// Mitsubishi GX Developer project: PLC_PCO520L2   PLC: Q06UDEH

PROGRAM ALARM
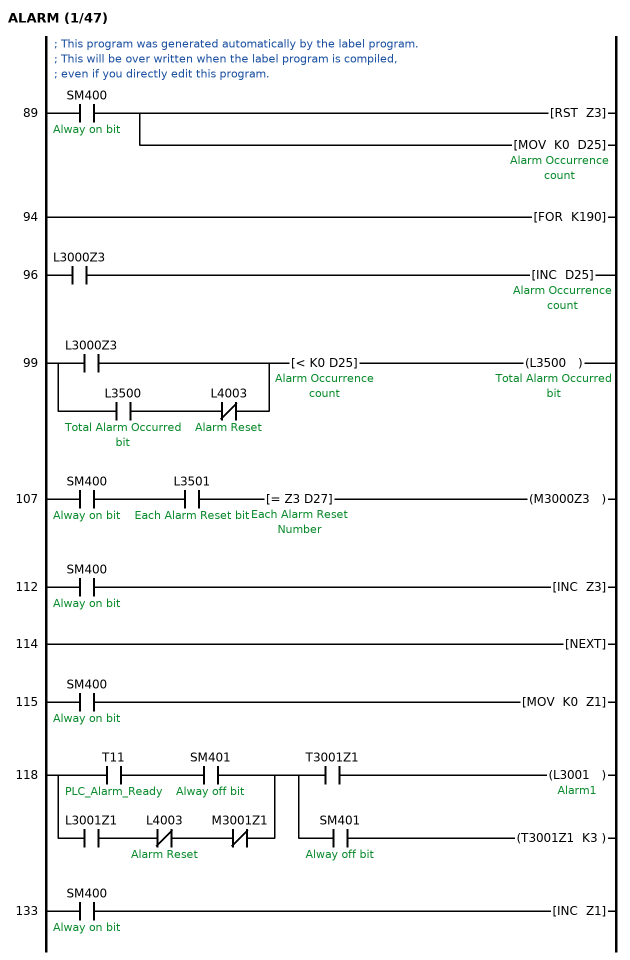
; This program was generated automatically by the label program.
; This will be over written when the label program is compiled,
; even if you directly edit this program.
89    LD      SM400  ; Alway on bit
      RST     Z3
      MOV     K0 D25  ; Alarm Occurrence count
94    FOR     K190
96    LD      L3000Z3
      INC     D25
99    LD      L3000Z3
      LD      L3500  ; Total Alarm Occurred bit
      ANI     L4003  ; Alarm Reset
      ORB
      AND<    K0 D25  ; Alarm Occurrence count
      OUT     L3500  ; Total Alarm Occurred bit
107   LD      SM400  ; Alway on bit
      AND     L3501  ; Each Alarm Reset bit
      AND=    Z3 D27  ; Each Alarm Reset Number
      OUT     M3000Z3
112   LD      SM400  ; Alway on bit
      INC     Z3
114   NEXT
115   LD      SM400  ; Alway on bit
      MOV     K0 Z1
118   LD      T11  ; PLC_Alarm_Ready
      AND     SM401  ; Alway off bit
      LD      L3001Z1
      ANI     L4003  ; Alarm Reset
      ANI     M3001Z1
      ORB
      MPS
      AND     T3001Z1
      OUT     L3001  ; Alarm1
      MPP
      AND     SM401  ; Alway off bit
      OUT     T3001Z1 K3
133   LD      SM400  ; Alway on bit
      INC     Z1
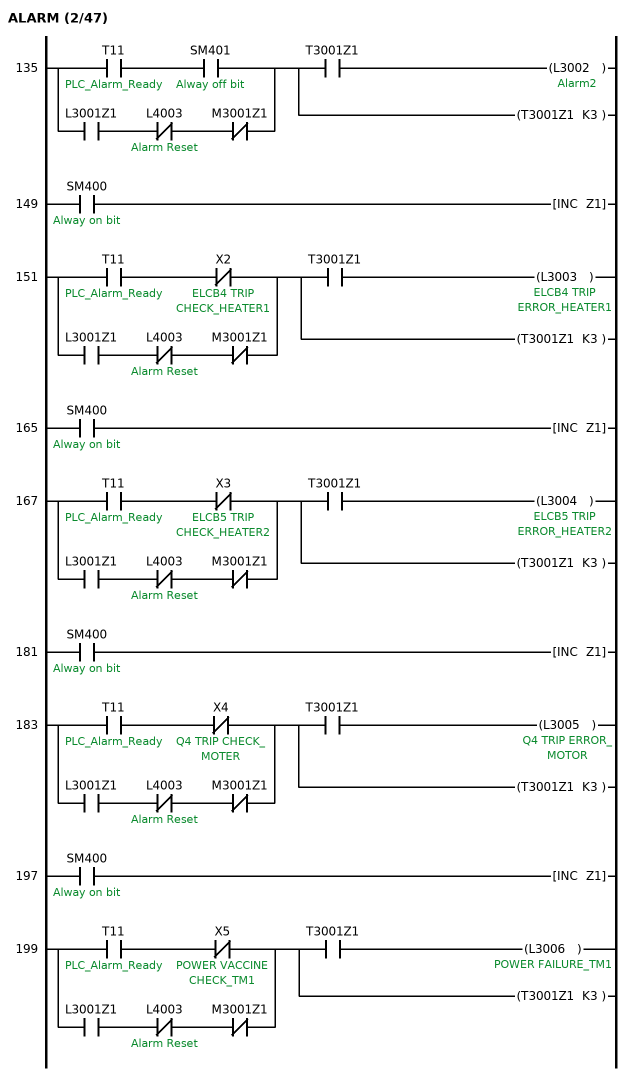
135   LD      T11  ; PLC_Alarm_Ready
      AND     SM401  ; Alway off bit
      LD      L3001Z1
      ANI     L4003  ; Alarm Reset
      ANI     M3001Z1
      ORB
      MPS
      AND     T3001Z1
      OUT     L3002  ; Alarm2
      MPP
      OUT     T3001Z1 K3
149   LD      SM400  ; Alway on bit
      INC     Z1
151   LD      T11  ; PLC_Alarm_Ready
      ANI     X2  ; ELCB4 TRIP CHECK_HEATER1
      LD      L3001Z1
      ANI     L4003  ; Alarm Reset
      ANI     M3001Z1
      ORB
      MPS
      AND     T3001Z1
      OUT     L3003  ; ELCB4 TRIP ERROR_HEATER1
      MPP
      OUT     T3001Z1 K3
165   LD      SM400  ; Alway on bit
      INC     Z1
167   LD      T11  ; PLC_Alarm_Ready
      ANI     X3  ; ELCB5 TRIP CHECK_HEATER2
      LD      L3001Z1
      ANI     L4003  ; Alarm Reset
      ANI     M3001Z1
      ORB
      MPS
      AND     T3001Z1
      OUT     L3004  ; ELCB5 TRIP ERROR_HEATER2
      MPP
      OUT     T3001Z1 K3
181   LD      SM400  ; Alway on bit
      INC     Z1
183   LD      T11  ; PLC_Alarm_Ready
      ANI     X4  ; Q4 TRIP CHECK_MOTER
      LD      L3001Z1
      ANI     L4003  ; Alarm Reset
      ANI     M3001Z1
      ORB
      MPS
      AND     T3001Z1
      OUT     L3005  ; Q4 TRIP ERROR_MOTOR
      MPP
      OUT     T3001Z1 K3
197   LD      SM400  ; Alway on bit
      INC     Z1
199   LD      T11  ; PLC_Alarm_Ready
      ANI     X5  ; POWER VACCINE CHECK_TM1
      LD      L3001Z1
      ANI     L4003  ; Alarm Reset
      ANI     M3001Z1
      ORB
      MPS
      AND     T3001Z1
      OUT     L3006  ; POWER FAILURE_TM1
      MPP
      OUT     T3001Z1 K3
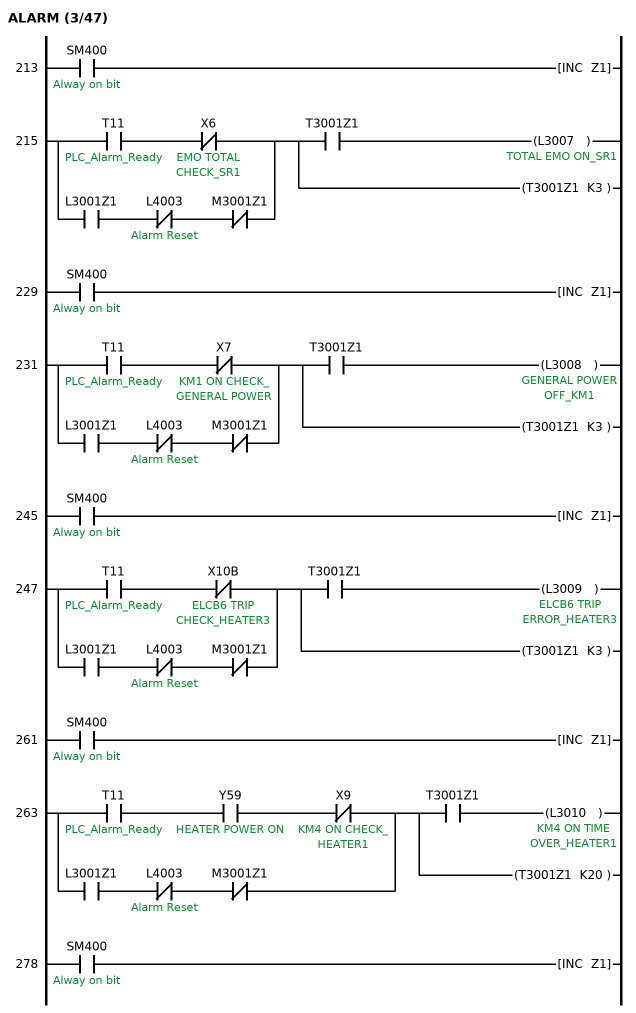
213   LD      SM400  ; Alway on bit
      INC     Z1
215   LD      T11  ; PLC_Alarm_Ready
      ANI     X6  ; EMO TOTAL CHECK_SR1
      LD      L3001Z1
      ANI     L4003  ; Alarm Reset
      ANI     M3001Z1
      ORB
      MPS
      AND     T3001Z1
      OUT     L3007  ; TOTAL EMO ON_SR1
      MPP
      OUT     T3001Z1 K3
229   LD      SM400  ; Alway on bit
      INC     Z1
231   LD      T11  ; PLC_Alarm_Ready
      ANI     X7  ; KM1 ON CHECK_GENERAL POWER
      LD      L3001Z1
      ANI     L4003  ; Alarm Reset
      ANI     M3001Z1
      ORB
      MPS
      AND     T3001Z1
      OUT     L3008  ; GENERAL POWER OFF_KM1
      MPP
      OUT     T3001Z1 K3
245   LD      SM400  ; Alway on bit
      INC     Z1
247   LD      T11  ; PLC_Alarm_Ready
      ANI     X10B  ; ELCB6 TRIP CHECK_HEATER3
      LD      L3001Z1
      ANI     L4003  ; Alarm Reset
      ANI     M3001Z1
      ORB
      MPS
      AND     T3001Z1
      OUT     L3009  ; ELCB6 TRIP ERROR_HEATER3
      MPP
      OUT     T3001Z1 K3
261   LD      SM400  ; Alway on bit
      INC     Z1
263   LD      T11  ; PLC_Alarm_Ready
      AND     Y59  ; HEATER POWER ON
      ANI     X9  ; KM4 ON CHECK_HEATER1
      LD      L3001Z1
      ANI     L4003  ; Alarm Reset
      ANI     M3001Z1
      ORB
      MPS
      AND     T3001Z1
      OUT     L3010  ; KM4 ON TIME OVER_HEATER1
      MPP
      OUT     T3001Z1 K20
278   LD      SM400  ; Alway on bit
      INC     Z1
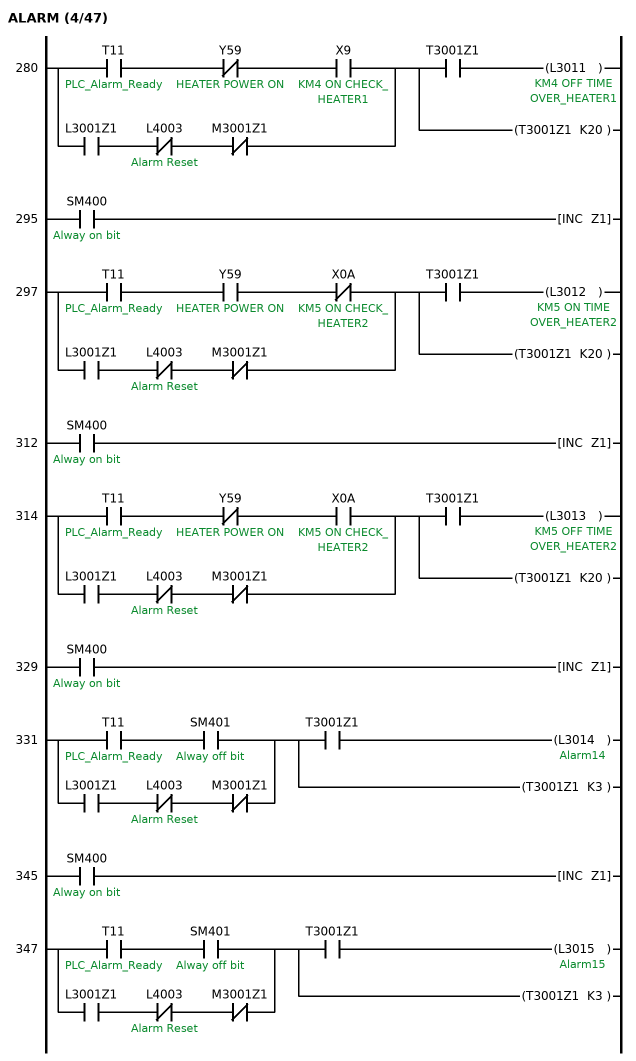
280   LD      T11  ; PLC_Alarm_Ready
      ANI     Y59  ; HEATER POWER ON
      AND     X9  ; KM4 ON CHECK_HEATER1
      LD      L3001Z1
      ANI     L4003  ; Alarm Reset
      ANI     M3001Z1
      ORB
      MPS
      AND     T3001Z1
      OUT     L3011  ; KM4 OFF TIME OVER_HEATER1
      MPP
      OUT     T3001Z1 K20
295   LD      SM400  ; Alway on bit
      INC     Z1
297   LD      T11  ; PLC_Alarm_Ready
      AND     Y59  ; HEATER POWER ON
      ANI     X0A  ; KM5 ON CHECK_HEATER2
      LD      L3001Z1
      ANI     L4003  ; Alarm Reset
      ANI     M3001Z1
      ORB
      MPS
      AND     T3001Z1
      OUT     L3012  ; KM5 ON TIME OVER_HEATER2
      MPP
      OUT     T3001Z1 K20
312   LD      SM400  ; Alway on bit
      INC     Z1
314   LD      T11  ; PLC_Alarm_Ready
      ANI     Y59  ; HEATER POWER ON
      AND     X0A  ; KM5 ON CHECK_HEATER2
      LD      L3001Z1
      ANI     L4003  ; Alarm Reset
      ANI     M3001Z1
      ORB
      MPS
      AND     T3001Z1
      OUT     L3013  ; KM5 OFF TIME OVER_HEATER2
      MPP
      OUT     T3001Z1 K20
329   LD      SM400  ; Alway on bit
      INC     Z1
331   LD      T11  ; PLC_Alarm_Ready
      AND     SM401  ; Alway off bit
      LD      L3001Z1
      ANI     L4003  ; Alarm Reset
      ANI     M3001Z1
      ORB
      MPS
      AND     T3001Z1
      OUT     L3014  ; Alarm14
      MPP
      OUT     T3001Z1 K3
345   LD      SM400  ; Alway on bit
      INC     Z1
347   LD      T11  ; PLC_Alarm_Ready
      AND     SM401  ; Alway off bit
      LD      L3001Z1
      ANI     L4003  ; Alarm Reset
      ANI     M3001Z1
      ORB
      MPS
      AND     T3001Z1
      OUT     L3015  ; Alarm15
      MPP
      OUT     T3001Z1 K3
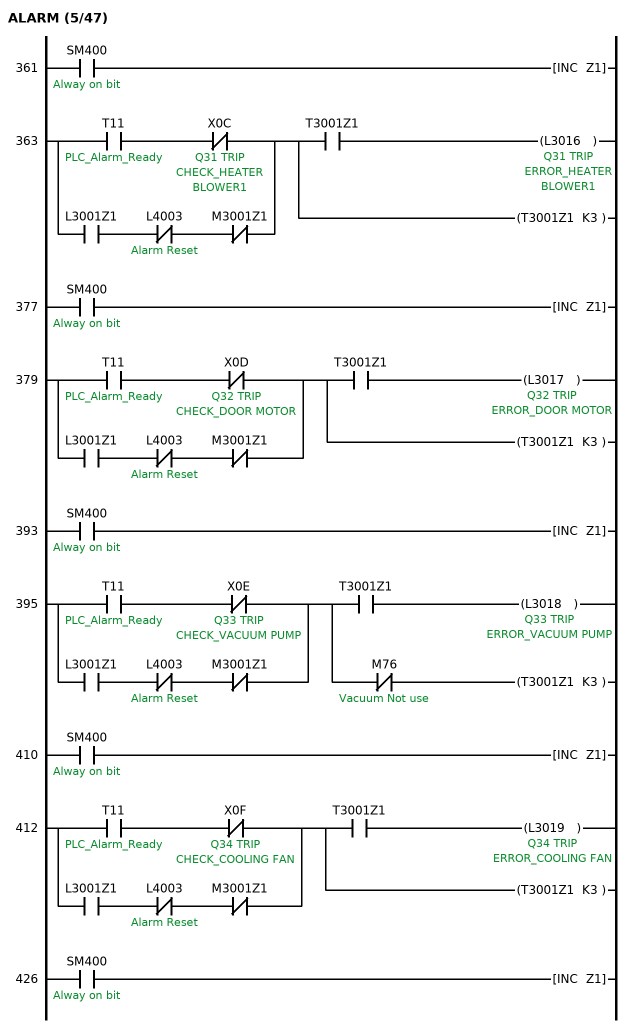
361   LD      SM400  ; Alway on bit
      INC     Z1
363   LD      T11  ; PLC_Alarm_Ready
      ANI     X0C  ; Q31 TRIP CHECK_HEATER BLOWER1
      LD      L3001Z1
      ANI     L4003  ; Alarm Reset
      ANI     M3001Z1
      ORB
      MPS
      AND     T3001Z1
      OUT     L3016  ; Q31 TRIP ERROR_HEATER BLOWER1
      MPP
      OUT     T3001Z1 K3
377   LD      SM400  ; Alway on bit
      INC     Z1
379   LD      T11  ; PLC_Alarm_Ready
      ANI     X0D  ; Q32 TRIP CHECK_DOOR MOTOR
      LD      L3001Z1
      ANI     L4003  ; Alarm Reset
      ANI     M3001Z1
      ORB
      MPS
      AND     T3001Z1
      OUT     L3017  ; Q32 TRIP ERROR_DOOR MOTOR
      MPP
      OUT     T3001Z1 K3
393   LD      SM400  ; Alway on bit
      INC     Z1
395   LD      T11  ; PLC_Alarm_Ready
      ANI     X0E  ; Q33 TRIP CHECK_VACUUM PUMP
      LD      L3001Z1
      ANI     L4003  ; Alarm Reset
      ANI     M3001Z1
      ORB
      MPS
      AND     T3001Z1
      OUT     L3018  ; Q33 TRIP ERROR_VACUUM PUMP
      MPP
      ANI     M76  ; Vacuum Not use
      OUT     T3001Z1 K3
410   LD      SM400  ; Alway on bit
      INC     Z1
412   LD      T11  ; PLC_Alarm_Ready
      ANI     X0F  ; Q34 TRIP CHECK_COOLING FAN
      LD      L3001Z1
      ANI     L4003  ; Alarm Reset
      ANI     M3001Z1
      ORB
      MPS
      AND     T3001Z1
      OUT     L3019  ; Q34 TRIP ERROR_COOLING FAN
      MPP
      OUT     T3001Z1 K3
426   LD      SM400  ; Alway on bit
      INC     Z1
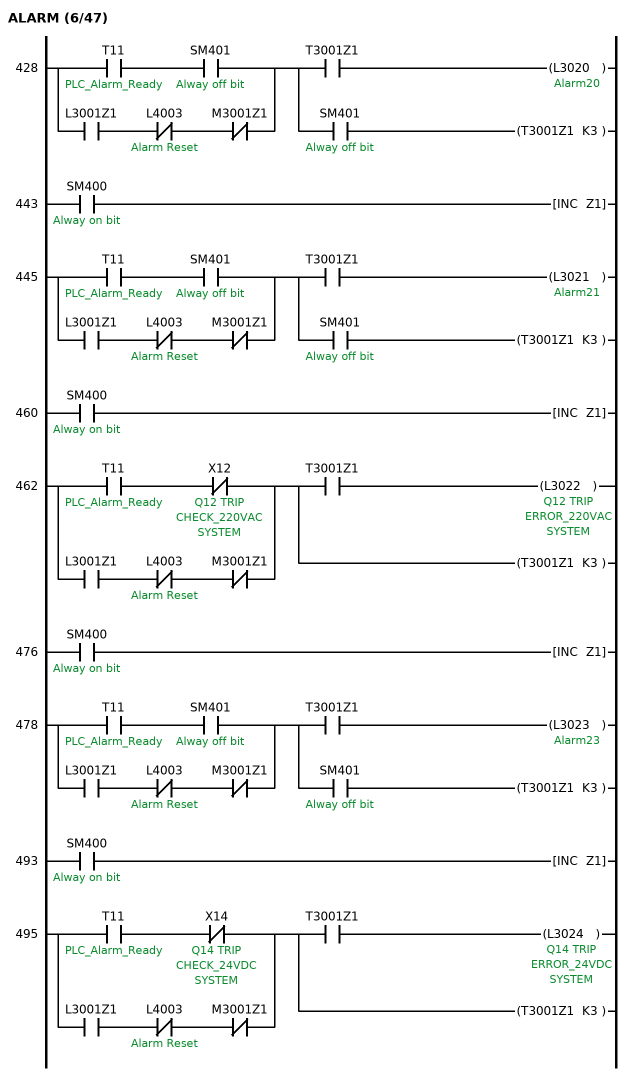
428   LD      T11  ; PLC_Alarm_Ready
      AND     SM401  ; Alway off bit
      LD      L3001Z1
      ANI     L4003  ; Alarm Reset
      ANI     M3001Z1
      ORB
      MPS
      AND     T3001Z1
      OUT     L3020  ; Alarm20
      MPP
      AND     SM401  ; Alway off bit
      OUT     T3001Z1 K3
443   LD      SM400  ; Alway on bit
      INC     Z1
445   LD      T11  ; PLC_Alarm_Ready
      AND     SM401  ; Alway off bit
      LD      L3001Z1
      ANI     L4003  ; Alarm Reset
      ANI     M3001Z1
      ORB
      MPS
      AND     T3001Z1
      OUT     L3021  ; Alarm21
      MPP
      AND     SM401  ; Alway off bit
      OUT     T3001Z1 K3
460   LD      SM400  ; Alway on bit
      INC     Z1
462   LD      T11  ; PLC_Alarm_Ready
      ANI     X12  ; Q12 TRIP CHECK_220VAC SYSTEM
      LD      L3001Z1
      ANI     L4003  ; Alarm Reset
      ANI     M3001Z1
      ORB
      MPS
      AND     T3001Z1
      OUT     L3022  ; Q12 TRIP ERROR_220VAC SYSTEM
      MPP
      OUT     T3001Z1 K3
476   LD      SM400  ; Alway on bit
      INC     Z1
478   LD      T11  ; PLC_Alarm_Ready
      AND     SM401  ; Alway off bit
      LD      L3001Z1
      ANI     L4003  ; Alarm Reset
      ANI     M3001Z1
      ORB
      MPS
      AND     T3001Z1
      OUT     L3023  ; Alarm23
      MPP
      AND     SM401  ; Alway off bit
      OUT     T3001Z1 K3
493   LD      SM400  ; Alway on bit
      INC     Z1
495   LD      T11  ; PLC_Alarm_Ready
      ANI     X14  ; Q14 TRIP CHECK_24VDC SYSTEM
      LD      L3001Z1
      ANI     L4003  ; Alarm Reset
      ANI     M3001Z1
      ORB
      MPS
      AND     T3001Z1
      OUT     L3024  ; Q14 TRIP ERROR_24VDC SYSTEM
      MPP
      OUT     T3001Z1 K3
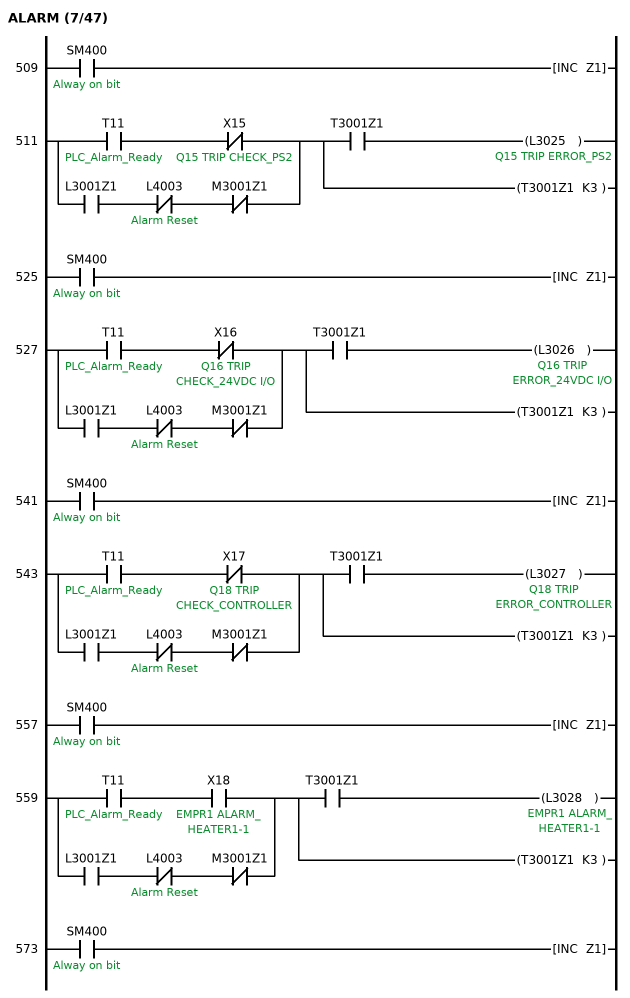
509   LD      SM400  ; Alway on bit
      INC     Z1
511   LD      T11  ; PLC_Alarm_Ready
      ANI     X15  ; Q15 TRIP CHECK_PS2
      LD      L3001Z1
      ANI     L4003  ; Alarm Reset
      ANI     M3001Z1
      ORB
      MPS
      AND     T3001Z1
      OUT     L3025  ; Q15 TRIP ERROR_PS2
      MPP
      OUT     T3001Z1 K3
525   LD      SM400  ; Alway on bit
      INC     Z1
527   LD      T11  ; PLC_Alarm_Ready
      ANI     X16  ; Q16 TRIP CHECK_24VDC I/O
      LD      L3001Z1
      ANI     L4003  ; Alarm Reset
      ANI     M3001Z1
      ORB
      MPS
      AND     T3001Z1
      OUT     L3026  ; Q16 TRIP ERROR_24VDC I/O
      MPP
      OUT     T3001Z1 K3
541   LD      SM400  ; Alway on bit
      INC     Z1
543   LD      T11  ; PLC_Alarm_Ready
      ANI     X17  ; Q18 TRIP CHECK_CONTROLLER
      LD      L3001Z1
      ANI     L4003  ; Alarm Reset
      ANI     M3001Z1
      ORB
      MPS
      AND     T3001Z1
      OUT     L3027  ; Q18 TRIP ERROR_CONTROLLER
      MPP
      OUT     T3001Z1 K3
557   LD      SM400  ; Alway on bit
      INC     Z1
559   LD      T11  ; PLC_Alarm_Ready
      AND     X18  ; EMPR1 ALARM_HEATER1-1
      LD      L3001Z1
      ANI     L4003  ; Alarm Reset
      ANI     M3001Z1
      ORB
      MPS
      AND     T3001Z1
      OUT     L3028  ; EMPR1 ALARM_HEATER1-1
      MPP
      OUT     T3001Z1 K3
573   LD      SM400  ; Alway on bit
      INC     Z1
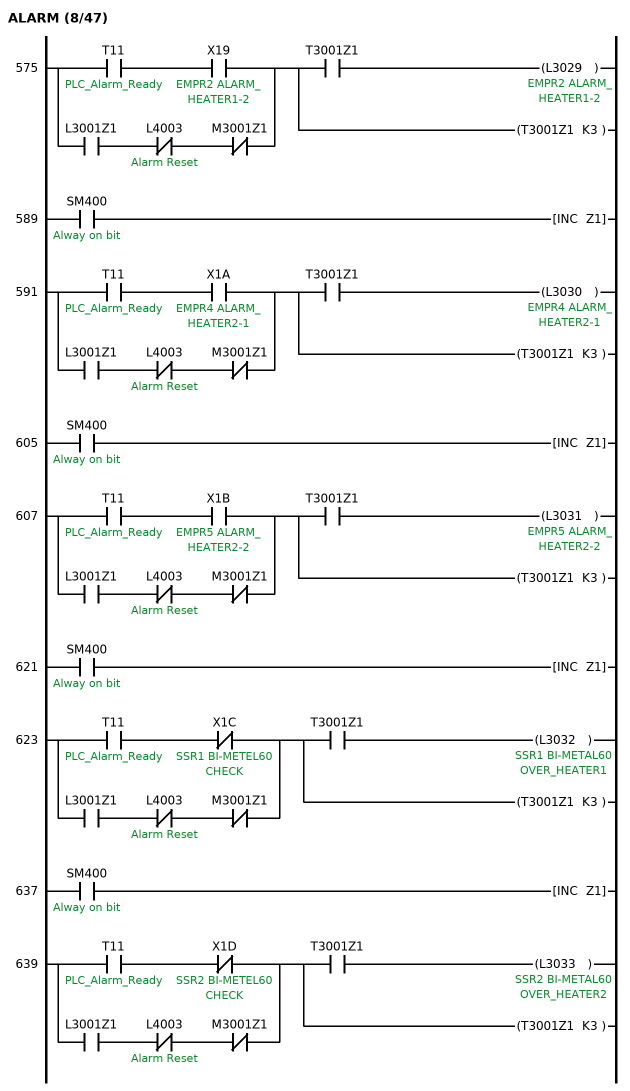
575   LD      T11  ; PLC_Alarm_Ready
      AND     X19  ; EMPR2 ALARM_HEATER1-2
      LD      L3001Z1
      ANI     L4003  ; Alarm Reset
      ANI     M3001Z1
      ORB
      MPS
      AND     T3001Z1
      OUT     L3029  ; EMPR2 ALARM_HEATER1-2
      MPP
      OUT     T3001Z1 K3
589   LD      SM400  ; Alway on bit
      INC     Z1
591   LD      T11  ; PLC_Alarm_Ready
      AND     X1A  ; EMPR4 ALARM_HEATER2-1
      LD      L3001Z1
      ANI     L4003  ; Alarm Reset
      ANI     M3001Z1
      ORB
      MPS
      AND     T3001Z1
      OUT     L3030  ; EMPR4 ALARM_HEATER2-1
      MPP
      OUT     T3001Z1 K3
605   LD      SM400  ; Alway on bit
      INC     Z1
607   LD      T11  ; PLC_Alarm_Ready
      AND     X1B  ; EMPR5 ALARM_HEATER2-2
      LD      L3001Z1
      ANI     L4003  ; Alarm Reset
      ANI     M3001Z1
      ORB
      MPS
      AND     T3001Z1
      OUT     L3031  ; EMPR5 ALARM_HEATER2-2
      MPP
      OUT     T3001Z1 K3
621   LD      SM400  ; Alway on bit
      INC     Z1
623   LD      T11  ; PLC_Alarm_Ready
      ANI     X1C  ; SSR1 BI-METEL60 CHECK
      LD      L3001Z1
      ANI     L4003  ; Alarm Reset
      ANI     M3001Z1
      ORB
      MPS
      AND     T3001Z1
      OUT     L3032  ; SSR1 BI-METAL60 OVER_HEATER1
      MPP
      OUT     T3001Z1 K3
637   LD      SM400  ; Alway on bit
      INC     Z1
639   LD      T11  ; PLC_Alarm_Ready
      ANI     X1D  ; SSR2 BI-METEL60 CHECK
      LD      L3001Z1
      ANI     L4003  ; Alarm Reset
      ANI     M3001Z1
      ORB
      MPS
      AND     T3001Z1
      OUT     L3033  ; SSR2 BI-METAL60 OVER_HEATER2
      MPP
      OUT     T3001Z1 K3
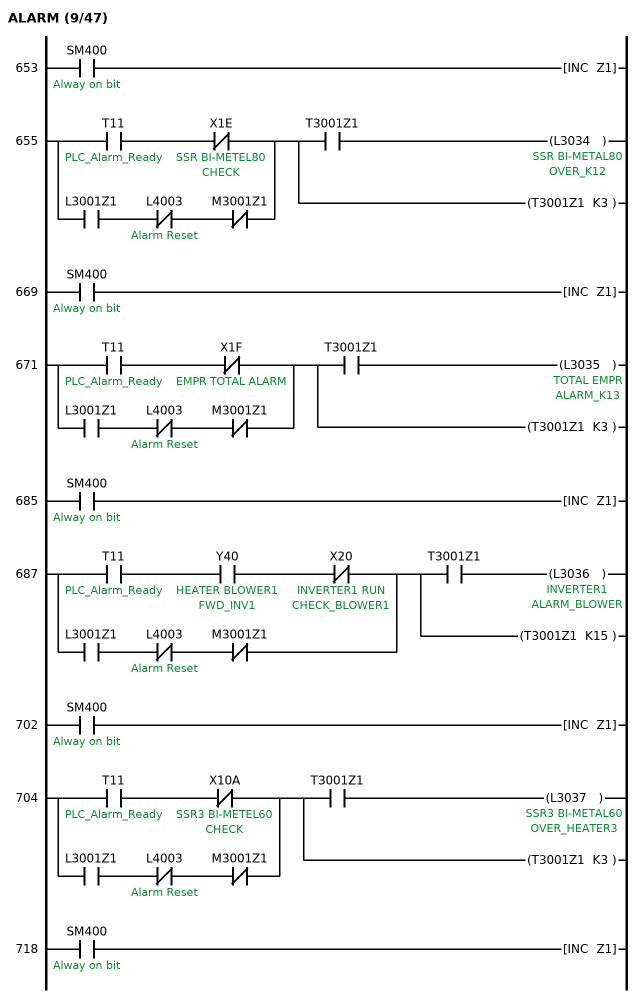
653   LD      SM400  ; Alway on bit
      INC     Z1
655   LD      T11  ; PLC_Alarm_Ready
      ANI     X1E  ; SSR BI-METEL80 CHECK
      LD      L3001Z1
      ANI     L4003  ; Alarm Reset
      ANI     M3001Z1
      ORB
      MPS
      AND     T3001Z1
      OUT     L3034  ; SSR BI-METAL80 OVER_K12
      MPP
      OUT     T3001Z1 K3
669   LD      SM400  ; Alway on bit
      INC     Z1
671   LD      T11  ; PLC_Alarm_Ready
      ANI     X1F  ; EMPR TOTAL ALARM
      LD      L3001Z1
      ANI     L4003  ; Alarm Reset
      ANI     M3001Z1
      ORB
      MPS
      AND     T3001Z1
      OUT     L3035  ; TOTAL EMPR ALARM_K13
      MPP
      OUT     T3001Z1 K3
685   LD      SM400  ; Alway on bit
      INC     Z1
687   LD      T11  ; PLC_Alarm_Ready
      AND     Y40  ; HEATER BLOWER1 FWD_INV1
      ANI     X20  ; INVERTER1 RUN CHECK_BLOWER1
      LD      L3001Z1
      ANI     L4003  ; Alarm Reset
      ANI     M3001Z1
      ORB
      MPS
      AND     T3001Z1
      OUT     L3036  ; INVERTER1 ALARM_BLOWER
      MPP
      OUT     T3001Z1 K15
702   LD      SM400  ; Alway on bit
      INC     Z1
704   LD      T11  ; PLC_Alarm_Ready
      ANI     X10A  ; SSR3 BI-METEL60 CHECK
      LD      L3001Z1
      ANI     L4003  ; Alarm Reset
      ANI     M3001Z1
      ORB
      MPS
      AND     T3001Z1
      OUT     L3037  ; SSR3 BI-METAL60 OVER_HEATER3
      MPP
      OUT     T3001Z1 K3
718   LD      SM400  ; Alway on bit
      INC     Z1
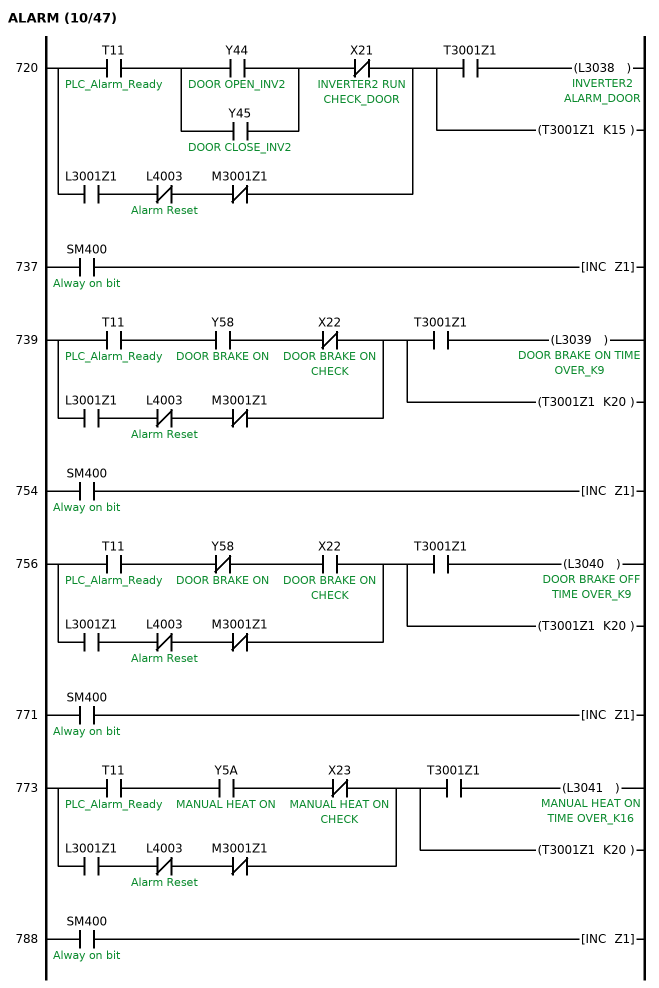
720   LD      T11  ; PLC_Alarm_Ready
      LD      Y44  ; DOOR OPEN_INV2
      OR      Y45  ; DOOR CLOSE_INV2
      ANB
      ANI     X21  ; INVERTER2 RUN CHECK_DOOR
      LD      L3001Z1
      ANI     L4003  ; Alarm Reset
      ANI     M3001Z1
      ORB
      MPS
      AND     T3001Z1
      OUT     L3038  ; INVERTER2 ALARM_DOOR
      MPP
      OUT     T3001Z1 K15
737   LD      SM400  ; Alway on bit
      INC     Z1
739   LD      T11  ; PLC_Alarm_Ready
      AND     Y58  ; DOOR BRAKE ON
      ANI     X22  ; DOOR BRAKE ON CHECK
      LD      L3001Z1
      ANI     L4003  ; Alarm Reset
      ANI     M3001Z1
      ORB
      MPS
      AND     T3001Z1
      OUT     L3039  ; DOOR BRAKE ON TIME OVER_K9
      MPP
      OUT     T3001Z1 K20
754   LD      SM400  ; Alway on bit
      INC     Z1
756   LD      T11  ; PLC_Alarm_Ready
      ANI     Y58  ; DOOR BRAKE ON
      AND     X22  ; DOOR BRAKE ON CHECK
      LD      L3001Z1
      ANI     L4003  ; Alarm Reset
      ANI     M3001Z1
      ORB
      MPS
      AND     T3001Z1
      OUT     L3040  ; DOOR BRAKE OFF TIME OVER_K9
      MPP
      OUT     T3001Z1 K20
771   LD      SM400  ; Alway on bit
      INC     Z1
773   LD      T11  ; PLC_Alarm_Ready
      AND     Y5A  ; MANUAL HEAT ON
      ANI     X23  ; MANUAL HEAT ON CHECK
      LD      L3001Z1
      ANI     L4003  ; Alarm Reset
      ANI     M3001Z1
      ORB
      MPS
      AND     T3001Z1
      OUT     L3041  ; MANUAL HEAT ON TIME OVER_K16
      MPP
      OUT     T3001Z1 K20
788   LD      SM400  ; Alway on bit
      INC     Z1
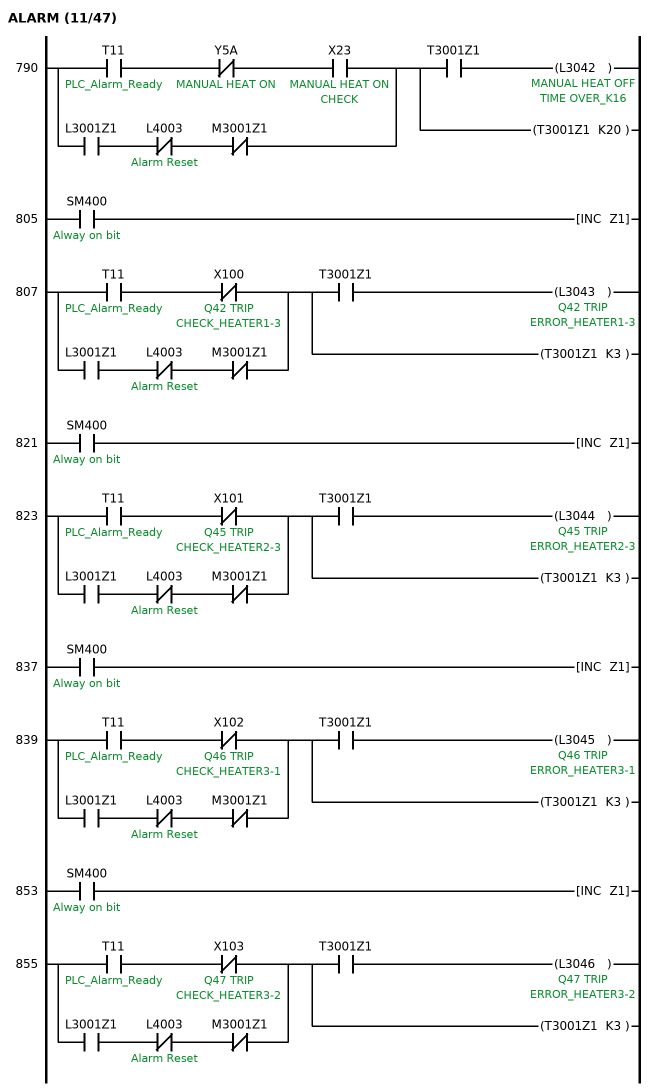
790   LD      T11  ; PLC_Alarm_Ready
      ANI     Y5A  ; MANUAL HEAT ON
      AND     X23  ; MANUAL HEAT ON CHECK
      LD      L3001Z1
      ANI     L4003  ; Alarm Reset
      ANI     M3001Z1
      ORB
      MPS
      AND     T3001Z1
      OUT     L3042  ; MANUAL HEAT OFF TIME OVER_K16
      MPP
      OUT     T3001Z1 K20
805   LD      SM400  ; Alway on bit
      INC     Z1
807   LD      T11  ; PLC_Alarm_Ready
      ANI     X100  ; Q42 TRIP CHECK_HEATER1-3
      LD      L3001Z1
      ANI     L4003  ; Alarm Reset
      ANI     M3001Z1
      ORB
      MPS
      AND     T3001Z1
      OUT     L3043  ; Q42 TRIP ERROR_HEATER1-3
      MPP
      OUT     T3001Z1 K3
821   LD      SM400  ; Alway on bit
      INC     Z1
823   LD      T11  ; PLC_Alarm_Ready
      ANI     X101  ; Q45 TRIP CHECK_HEATER2-3
      LD      L3001Z1
      ANI     L4003  ; Alarm Reset
      ANI     M3001Z1
      ORB
      MPS
      AND     T3001Z1
      OUT     L3044  ; Q45 TRIP ERROR_HEATER2-3
      MPP
      OUT     T3001Z1 K3
837   LD      SM400  ; Alway on bit
      INC     Z1
839   LD      T11  ; PLC_Alarm_Ready
      ANI     X102  ; Q46 TRIP CHECK_HEATER3-1
      LD      L3001Z1
      ANI     L4003  ; Alarm Reset
      ANI     M3001Z1
      ORB
      MPS
      AND     T3001Z1
      OUT     L3045  ; Q46 TRIP ERROR_HEATER3-1
      MPP
      OUT     T3001Z1 K3
853   LD      SM400  ; Alway on bit
      INC     Z1
855   LD      T11  ; PLC_Alarm_Ready
      ANI     X103  ; Q47 TRIP CHECK_HEATER3-2
      LD      L3001Z1
      ANI     L4003  ; Alarm Reset
      ANI     M3001Z1
      ORB
      MPS
      AND     T3001Z1
      OUT     L3046  ; Q47 TRIP ERROR_HEATER3-2
      MPP
      OUT     T3001Z1 K3
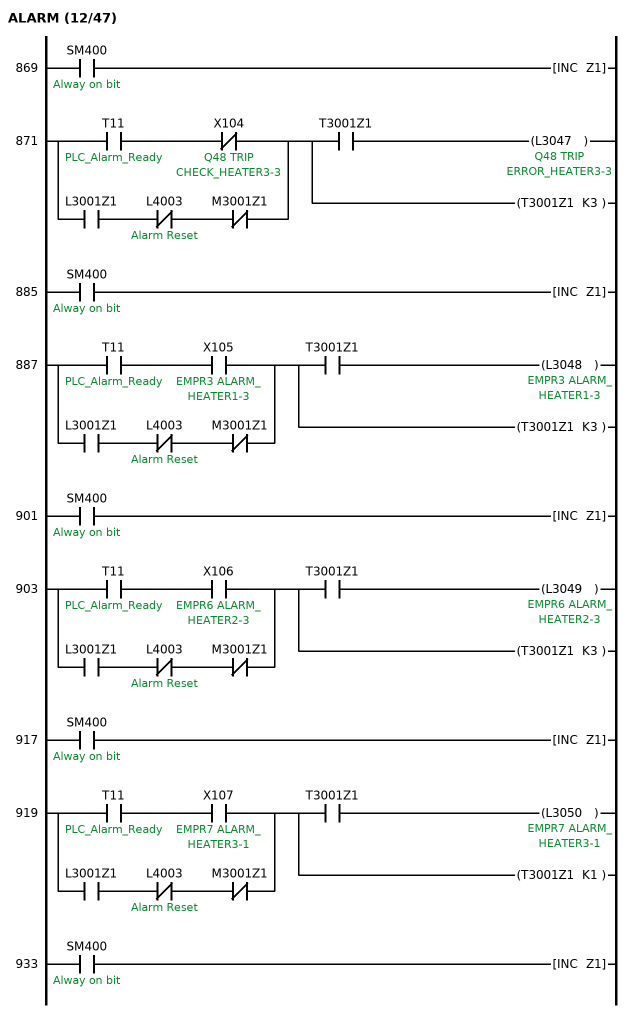
869   LD      SM400  ; Alway on bit
      INC     Z1
871   LD      T11  ; PLC_Alarm_Ready
      ANI     X104  ; Q48 TRIP CHECK_HEATER3-3
      LD      L3001Z1
      ANI     L4003  ; Alarm Reset
      ANI     M3001Z1
      ORB
      MPS
      AND     T3001Z1
      OUT     L3047  ; Q48 TRIP ERROR_HEATER3-3
      MPP
      OUT     T3001Z1 K3
885   LD      SM400  ; Alway on bit
      INC     Z1
887   LD      T11  ; PLC_Alarm_Ready
      AND     X105  ; EMPR3 ALARM_HEATER1-3
      LD      L3001Z1
      ANI     L4003  ; Alarm Reset
      ANI     M3001Z1
      ORB
      MPS
      AND     T3001Z1
      OUT     L3048  ; EMPR3 ALARM_HEATER1-3
      MPP
      OUT     T3001Z1 K3
901   LD      SM400  ; Alway on bit
      INC     Z1
903   LD      T11  ; PLC_Alarm_Ready
      AND     X106  ; EMPR6 ALARM_HEATER2-3
      LD      L3001Z1
      ANI     L4003  ; Alarm Reset
      ANI     M3001Z1
      ORB
      MPS
      AND     T3001Z1
      OUT     L3049  ; EMPR6 ALARM_HEATER2-3
      MPP
      OUT     T3001Z1 K3
917   LD      SM400  ; Alway on bit
      INC     Z1
919   LD      T11  ; PLC_Alarm_Ready
      AND     X107  ; EMPR7 ALARM_HEATER3-1
      LD      L3001Z1
      ANI     L4003  ; Alarm Reset
      ANI     M3001Z1
      ORB
      MPS
      AND     T3001Z1
      OUT     L3050  ; EMPR7 ALARM_HEATER3-1
      MPP
      OUT     T3001Z1 K1
933   LD      SM400  ; Alway on bit
      INC     Z1
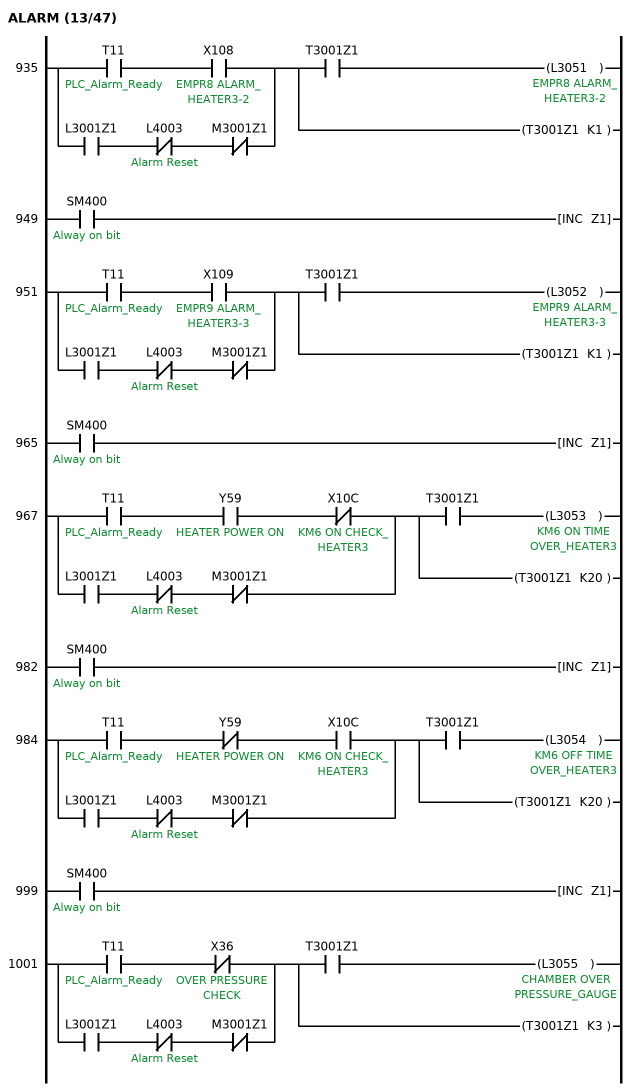
935   LD      T11  ; PLC_Alarm_Ready
      AND     X108  ; EMPR8 ALARM_HEATER3-2
      LD      L3001Z1
      ANI     L4003  ; Alarm Reset
      ANI     M3001Z1
      ORB
      MPS
      AND     T3001Z1
      OUT     L3051  ; EMPR8 ALARM_HEATER3-2
      MPP
      OUT     T3001Z1 K1
949   LD      SM400  ; Alway on bit
      INC     Z1
951   LD      T11  ; PLC_Alarm_Ready
      AND     X109  ; EMPR9 ALARM_HEATER3-3
      LD      L3001Z1
      ANI     L4003  ; Alarm Reset
      ANI     M3001Z1
      ORB
      MPS
      AND     T3001Z1
      OUT     L3052  ; EMPR9 ALARM_HEATER3-3
      MPP
      OUT     T3001Z1 K1
965   LD      SM400  ; Alway on bit
      INC     Z1
967   LD      T11  ; PLC_Alarm_Ready
      AND     Y59  ; HEATER POWER ON
      ANI     X10C  ; KM6 ON CHECK_HEATER3
      LD      L3001Z1
      ANI     L4003  ; Alarm Reset
      ANI     M3001Z1
      ORB
      MPS
      AND     T3001Z1
      OUT     L3053  ; KM6 ON TIME OVER_HEATER3
      MPP
      OUT     T3001Z1 K20
982   LD      SM400  ; Alway on bit
      INC     Z1
984   LD      T11  ; PLC_Alarm_Ready
      ANI     Y59  ; HEATER POWER ON
      AND     X10C  ; KM6 ON CHECK_HEATER3
      LD      L3001Z1
      ANI     L4003  ; Alarm Reset
      ANI     M3001Z1
      ORB
      MPS
      AND     T3001Z1
      OUT     L3054  ; KM6 OFF TIME OVER_HEATER3
      MPP
      OUT     T3001Z1 K20
999   LD      SM400  ; Alway on bit
      INC     Z1
1001  LD      T11  ; PLC_Alarm_Ready
      ANI     X36  ; OVER PRESSURE CHECK
      LD      L3001Z1
      ANI     L4003  ; Alarm Reset
      ANI     M3001Z1
      ORB
      MPS
      AND     T3001Z1
      OUT     L3055  ; CHAMBER OVER PRESSURE_GAUGE
      MPP
      OUT     T3001Z1 K3
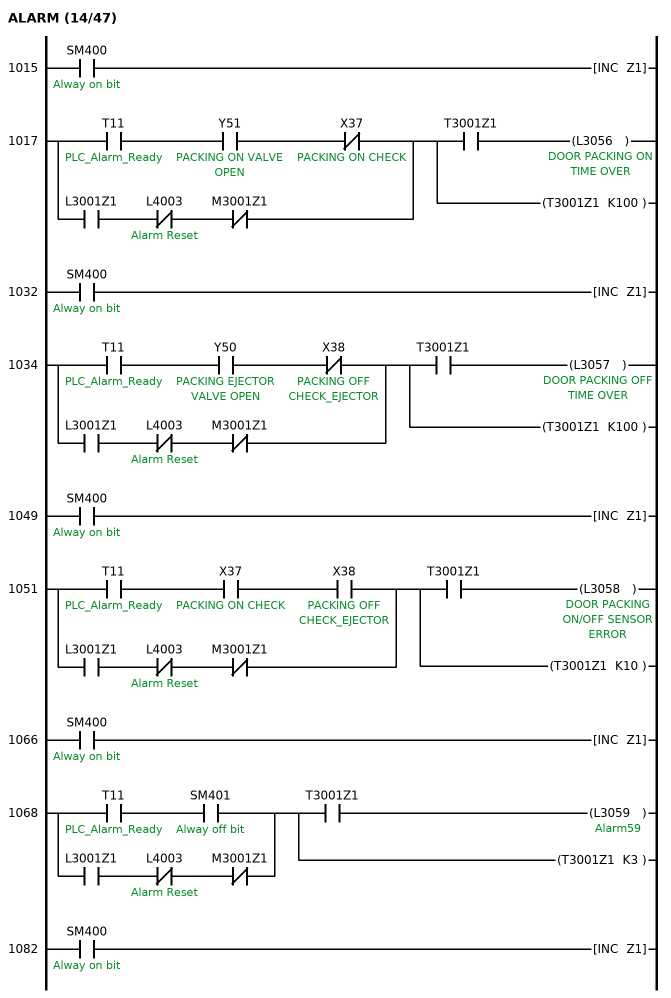
1015  LD      SM400  ; Alway on bit
      INC     Z1
1017  LD      T11  ; PLC_Alarm_Ready
      AND     Y51  ; PACKING ON VALVE OPEN
      ANI     X37  ; PACKING ON CHECK
      LD      L3001Z1
      ANI     L4003  ; Alarm Reset
      ANI     M3001Z1
      ORB
      MPS
      AND     T3001Z1
      OUT     L3056  ; DOOR PACKING ON TIME OVER
      MPP
      OUT     T3001Z1 K100
1032  LD      SM400  ; Alway on bit
      INC     Z1
1034  LD      T11  ; PLC_Alarm_Ready
      AND     Y50  ; PACKING EJECTOR VALVE OPEN
      ANI     X38  ; PACKING OFF CHECK_EJECTOR
      LD      L3001Z1
      ANI     L4003  ; Alarm Reset
      ANI     M3001Z1
      ORB
      MPS
      AND     T3001Z1
      OUT     L3057  ; DOOR PACKING OFF TIME OVER
      MPP
      OUT     T3001Z1 K100
1049  LD      SM400  ; Alway on bit
      INC     Z1
1051  LD      T11  ; PLC_Alarm_Ready
      AND     X37  ; PACKING ON CHECK
      AND     X38  ; PACKING OFF CHECK_EJECTOR
      LD      L3001Z1
      ANI     L4003  ; Alarm Reset
      ANI     M3001Z1
      ORB
      MPS
      AND     T3001Z1
      OUT     L3058  ; DOOR PACKING ON/OFF SENSOR ERROR
      MPP
      OUT     T3001Z1 K10
1066  LD      SM400  ; Alway on bit
      INC     Z1
1068  LD      T11  ; PLC_Alarm_Ready
      AND     SM401  ; Alway off bit
      LD      L3001Z1
      ANI     L4003  ; Alarm Reset
      ANI     M3001Z1
      ORB
      MPS
      AND     T3001Z1
      OUT     L3059  ; Alarm59
      MPP
      OUT     T3001Z1 K3
1082  LD      SM400  ; Alway on bit
      INC     Z1
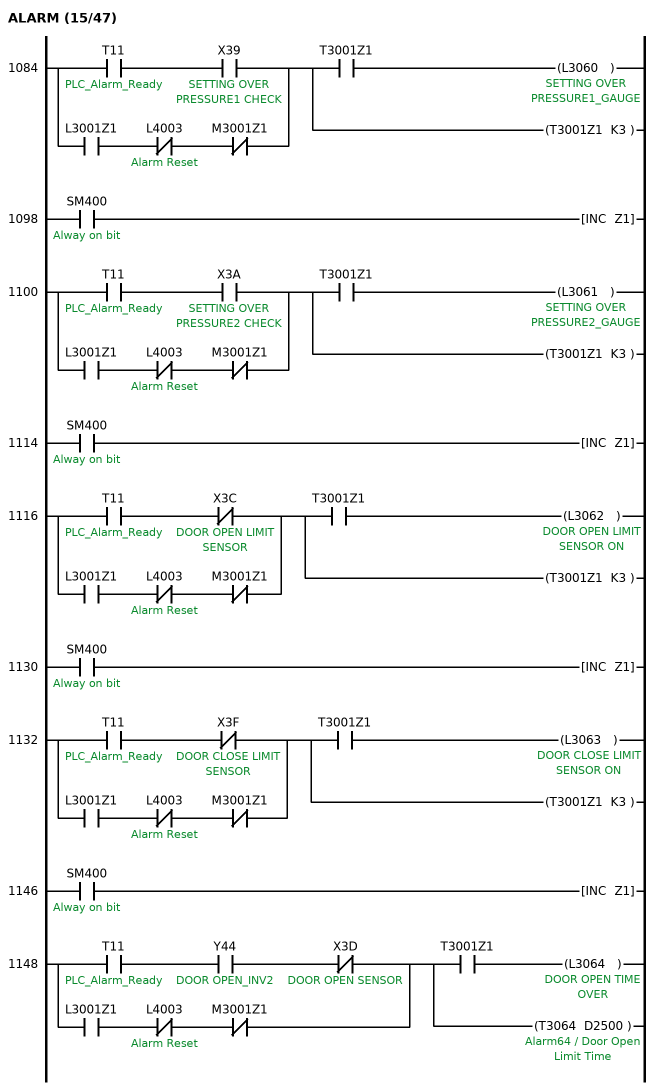
1084  LD      T11  ; PLC_Alarm_Ready
      AND     X39  ; SETTING OVER PRESSURE1 CHECK
      LD      L3001Z1
      ANI     L4003  ; Alarm Reset
      ANI     M3001Z1
      ORB
      MPS
      AND     T3001Z1
      OUT     L3060  ; SETTING OVER PRESSURE1_GAUGE
      MPP
      OUT     T3001Z1 K3
1098  LD      SM400  ; Alway on bit
      INC     Z1
1100  LD      T11  ; PLC_Alarm_Ready
      AND     X3A  ; SETTING OVER PRESSURE2 CHECK
      LD      L3001Z1
      ANI     L4003  ; Alarm Reset
      ANI     M3001Z1
      ORB
      MPS
      AND     T3001Z1
      OUT     L3061  ; SETTING OVER PRESSURE2_GAUGE
      MPP
      OUT     T3001Z1 K3
1114  LD      SM400  ; Alway on bit
      INC     Z1
1116  LD      T11  ; PLC_Alarm_Ready
      ANI     X3C  ; DOOR OPEN LIMIT SENSOR
      LD      L3001Z1
      ANI     L4003  ; Alarm Reset
      ANI     M3001Z1
      ORB
      MPS
      AND     T3001Z1
      OUT     L3062  ; DOOR OPEN LIMIT SENSOR ON
      MPP
      OUT     T3001Z1 K3
1130  LD      SM400  ; Alway on bit
      INC     Z1
1132  LD      T11  ; PLC_Alarm_Ready
      ANI     X3F  ; DOOR CLOSE LIMIT SENSOR
      LD      L3001Z1
      ANI     L4003  ; Alarm Reset
      ANI     M3001Z1
      ORB
      MPS
      AND     T3001Z1
      OUT     L3063  ; DOOR CLOSE LIMIT SENSOR ON
      MPP
      OUT     T3001Z1 K3
1146  LD      SM400  ; Alway on bit
      INC     Z1
1148  LD      T11  ; PLC_Alarm_Ready
      AND     Y44  ; DOOR OPEN_INV2
      ANI     X3D  ; DOOR OPEN SENSOR
      LD      L3001Z1
      ANI     L4003  ; Alarm Reset
      ANI     M3001Z1
      ORB
      MPS
      AND     T3001Z1
      OUT     L3064  ; DOOR OPEN TIME OVER
      MPP
      OUT     T3064 D2500  ; Alarm64 / Door Open Limit Time
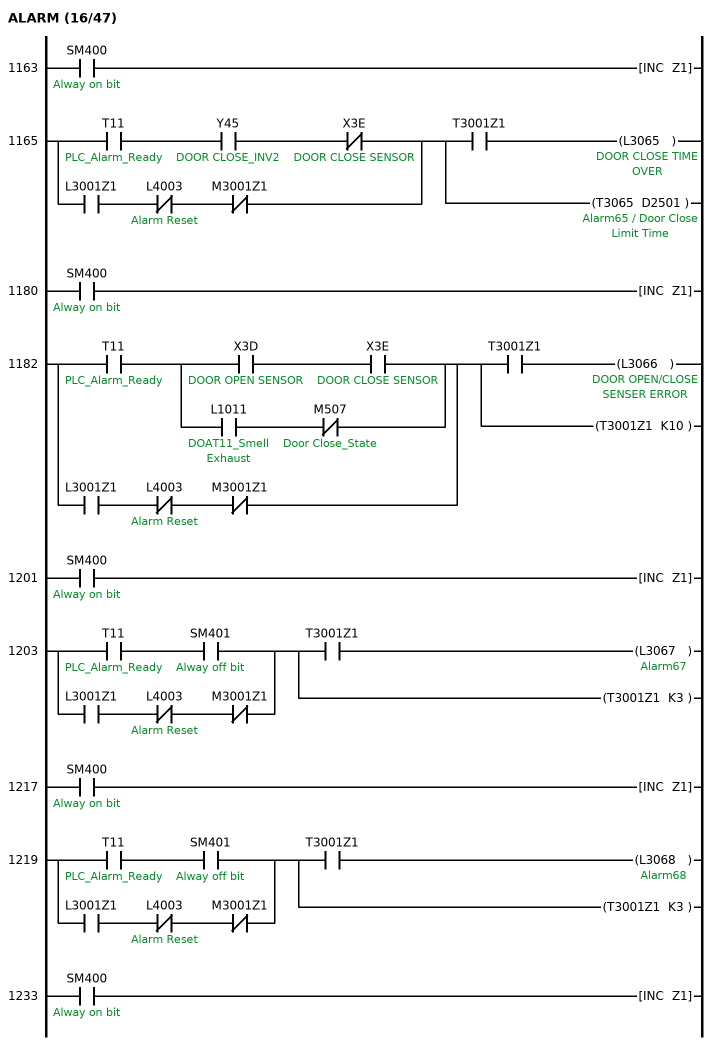
1163  LD      SM400  ; Alway on bit
      INC     Z1
1165  LD      T11  ; PLC_Alarm_Ready
      AND     Y45  ; DOOR CLOSE_INV2
      ANI     X3E  ; DOOR CLOSE SENSOR
      LD      L3001Z1
      ANI     L4003  ; Alarm Reset
      ANI     M3001Z1
      ORB
      MPS
      AND     T3001Z1
      OUT     L3065  ; DOOR CLOSE TIME OVER
      MPP
      OUT     T3065 D2501  ; Alarm65 / Door Close Limit Time
1180  LD      SM400  ; Alway on bit
      INC     Z1
1182  LD      T11  ; PLC_Alarm_Ready
      LD      X3D  ; DOOR OPEN SENSOR
      AND     X3E  ; DOOR CLOSE SENSOR
      LD      L1011  ; DOAT11_Smell Exhaust
      ANI     M507  ; Door Close_State
      ORB
      ANB
      LD      L3001Z1
      ANI     L4003  ; Alarm Reset
      ANI     M3001Z1
      ORB
      MPS
      AND     T3001Z1
      OUT     L3066  ; DOOR OPEN/CLOSE SENSER ERROR
      MPP
      OUT     T3001Z1 K10
1201  LD      SM400  ; Alway on bit
      INC     Z1
1203  LD      T11  ; PLC_Alarm_Ready
      AND     SM401  ; Alway off bit
      LD      L3001Z1
      ANI     L4003  ; Alarm Reset
      ANI     M3001Z1
      ORB
      MPS
      AND     T3001Z1
      OUT     L3067  ; Alarm67
      MPP
      OUT     T3001Z1 K3
1217  LD      SM400  ; Alway on bit
      INC     Z1
1219  LD      T11  ; PLC_Alarm_Ready
      AND     SM401  ; Alway off bit
      LD      L3001Z1
      ANI     L4003  ; Alarm Reset
      ANI     M3001Z1
      ORB
      MPS
      AND     T3001Z1
      OUT     L3068  ; Alarm68
      MPP
      OUT     T3001Z1 K3
1233  LD      SM400  ; Alway on bit
      INC     Z1
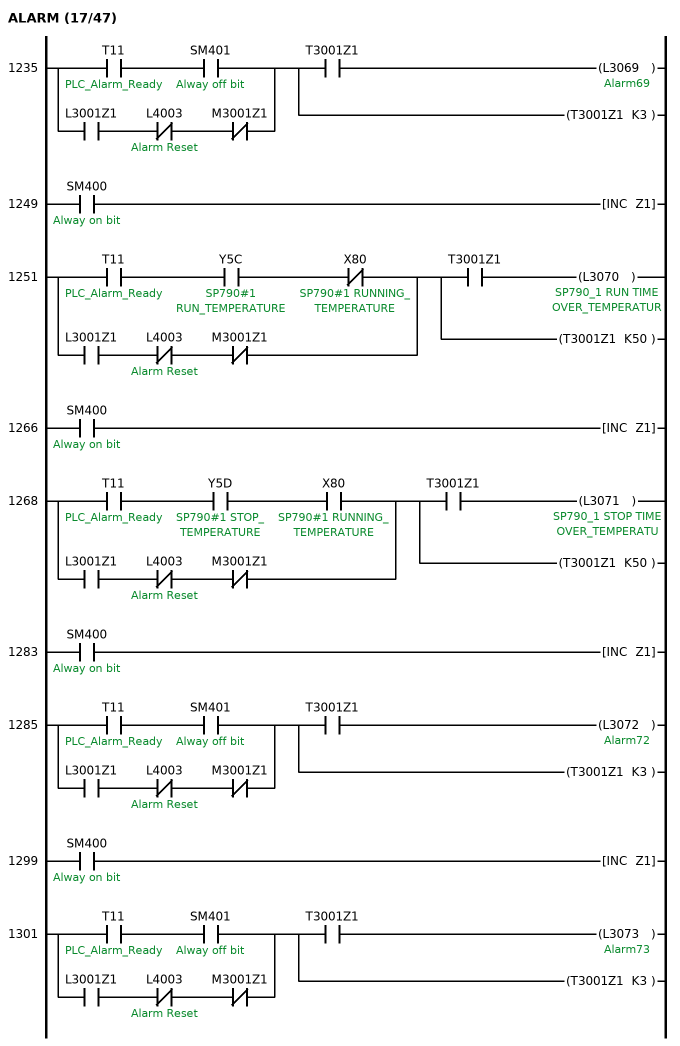
1235  LD      T11  ; PLC_Alarm_Ready
      AND     SM401  ; Alway off bit
      LD      L3001Z1
      ANI     L4003  ; Alarm Reset
      ANI     M3001Z1
      ORB
      MPS
      AND     T3001Z1
      OUT     L3069  ; Alarm69
      MPP
      OUT     T3001Z1 K3
1249  LD      SM400  ; Alway on bit
      INC     Z1
1251  LD      T11  ; PLC_Alarm_Ready
      AND     Y5C  ; SP790#1 RUN_TEMPERATURE
      ANI     X80  ; SP790#1 RUNNING_TEMPERATURE
      LD      L3001Z1
      ANI     L4003  ; Alarm Reset
      ANI     M3001Z1
      ORB
      MPS
      AND     T3001Z1
      OUT     L3070  ; SP790_1 RUN TIME OVER_TEMPERATUR
      MPP
      OUT     T3001Z1 K50
1266  LD      SM400  ; Alway on bit
      INC     Z1
1268  LD      T11  ; PLC_Alarm_Ready
      AND     Y5D  ; SP790#1 STOP_TEMPERATURE
      AND     X80  ; SP790#1 RUNNING_TEMPERATURE
      LD      L3001Z1
      ANI     L4003  ; Alarm Reset
      ANI     M3001Z1
      ORB
      MPS
      AND     T3001Z1
      OUT     L3071  ; SP790_1 STOP TIME OVER_TEMPERATU
      MPP
      OUT     T3001Z1 K50
1283  LD      SM400  ; Alway on bit
      INC     Z1
1285  LD      T11  ; PLC_Alarm_Ready
      AND     SM401  ; Alway off bit
      LD      L3001Z1
      ANI     L4003  ; Alarm Reset
      ANI     M3001Z1
      ORB
      MPS
      AND     T3001Z1
      OUT     L3072  ; Alarm72
      MPP
      OUT     T3001Z1 K3
1299  LD      SM400  ; Alway on bit
      INC     Z1
1301  LD      T11  ; PLC_Alarm_Ready
      AND     SM401  ; Alway off bit
      LD      L3001Z1
      ANI     L4003  ; Alarm Reset
      ANI     M3001Z1
      ORB
      MPS
      AND     T3001Z1
      OUT     L3073  ; Alarm73
      MPP
      OUT     T3001Z1 K3
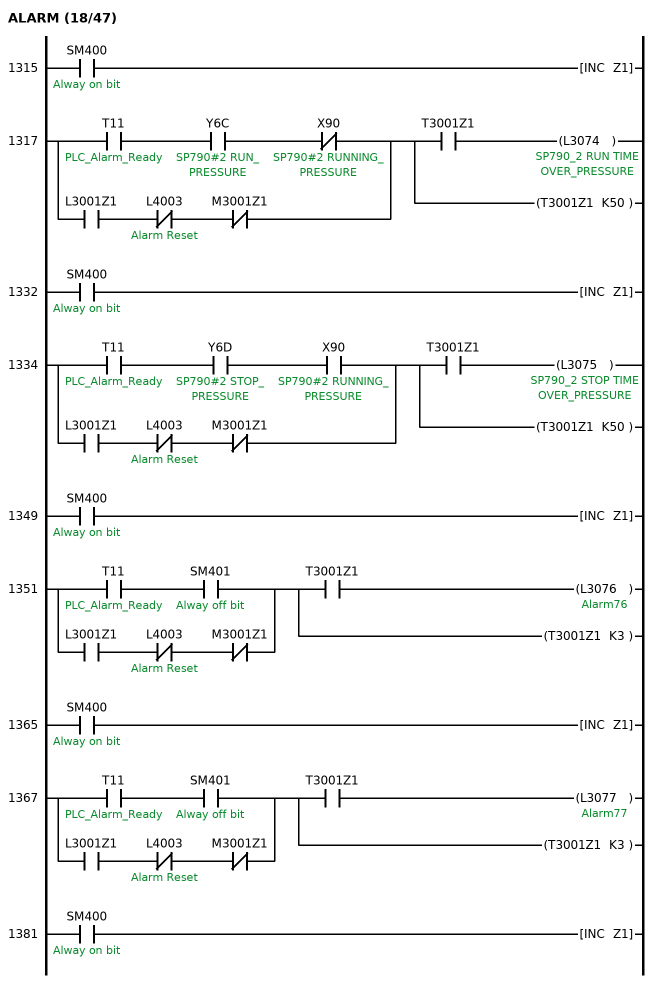
1315  LD      SM400  ; Alway on bit
      INC     Z1
1317  LD      T11  ; PLC_Alarm_Ready
      AND     Y6C  ; SP790#2 RUN_PRESSURE
      ANI     X90  ; SP790#2 RUNNING_PRESSURE
      LD      L3001Z1
      ANI     L4003  ; Alarm Reset
      ANI     M3001Z1
      ORB
      MPS
      AND     T3001Z1
      OUT     L3074  ; SP790_2 RUN TIME OVER_PRESSURE
      MPP
      OUT     T3001Z1 K50
1332  LD      SM400  ; Alway on bit
      INC     Z1
1334  LD      T11  ; PLC_Alarm_Ready
      AND     Y6D  ; SP790#2 STOP_PRESSURE
      AND     X90  ; SP790#2 RUNNING_PRESSURE
      LD      L3001Z1
      ANI     L4003  ; Alarm Reset
      ANI     M3001Z1
      ORB
      MPS
      AND     T3001Z1
      OUT     L3075  ; SP790_2 STOP TIME OVER_PRESSURE
      MPP
      OUT     T3001Z1 K50
1349  LD      SM400  ; Alway on bit
      INC     Z1
1351  LD      T11  ; PLC_Alarm_Ready
      AND     SM401  ; Alway off bit
      LD      L3001Z1
      ANI     L4003  ; Alarm Reset
      ANI     M3001Z1
      ORB
      MPS
      AND     T3001Z1
      OUT     L3076  ; Alarm76
      MPP
      OUT     T3001Z1 K3
1365  LD      SM400  ; Alway on bit
      INC     Z1
1367  LD      T11  ; PLC_Alarm_Ready
      AND     SM401  ; Alway off bit
      LD      L3001Z1
      ANI     L4003  ; Alarm Reset
      ANI     M3001Z1
      ORB
      MPS
      AND     T3001Z1
      OUT     L3077  ; Alarm77
      MPP
      OUT     T3001Z1 K3
1381  LD      SM400  ; Alway on bit
      INC     Z1
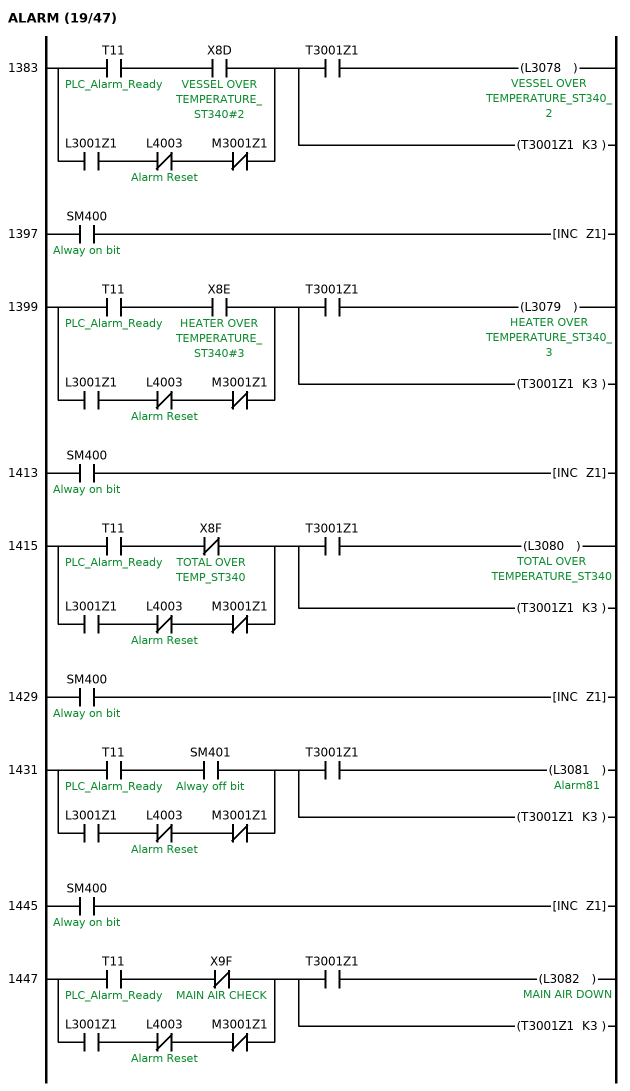
1383  LD      T11  ; PLC_Alarm_Ready
      AND     X8D  ; VESSEL OVER TEMPERATURE_ST340#2
      LD      L3001Z1
      ANI     L4003  ; Alarm Reset
      ANI     M3001Z1
      ORB
      MPS
      AND     T3001Z1
      OUT     L3078  ; VESSEL OVER TEMPERATURE_ST340_2
      MPP
      OUT     T3001Z1 K3
1397  LD      SM400  ; Alway on bit
      INC     Z1
1399  LD      T11  ; PLC_Alarm_Ready
      AND     X8E  ; HEATER OVER TEMPERATURE_ST340#3
      LD      L3001Z1
      ANI     L4003  ; Alarm Reset
      ANI     M3001Z1
      ORB
      MPS
      AND     T3001Z1
      OUT     L3079  ; HEATER OVER TEMPERATURE_ST340_3
      MPP
      OUT     T3001Z1 K3
1413  LD      SM400  ; Alway on bit
      INC     Z1
1415  LD      T11  ; PLC_Alarm_Ready
      ANI     X8F  ; TOTAL OVER TEMP_ST340
      LD      L3001Z1
      ANI     L4003  ; Alarm Reset
      ANI     M3001Z1
      ORB
      MPS
      AND     T3001Z1
      OUT     L3080  ; TOTAL OVER TEMPERATURE_ST340
      MPP
      OUT     T3001Z1 K3
1429  LD      SM400  ; Alway on bit
      INC     Z1
1431  LD      T11  ; PLC_Alarm_Ready
      AND     SM401  ; Alway off bit
      LD      L3001Z1
      ANI     L4003  ; Alarm Reset
      ANI     M3001Z1
      ORB
      MPS
      AND     T3001Z1
      OUT     L3081  ; Alarm81
      MPP
      OUT     T3001Z1 K3
1445  LD      SM400  ; Alway on bit
      INC     Z1
1447  LD      T11  ; PLC_Alarm_Ready
      ANI     X9F  ; MAIN AIR CHECK
      LD      L3001Z1
      ANI     L4003  ; Alarm Reset
      ANI     M3001Z1
      ORB
      MPS
      AND     T3001Z1
      OUT     L3082  ; MAIN AIR DOWN
      MPP
      OUT     T3001Z1 K3
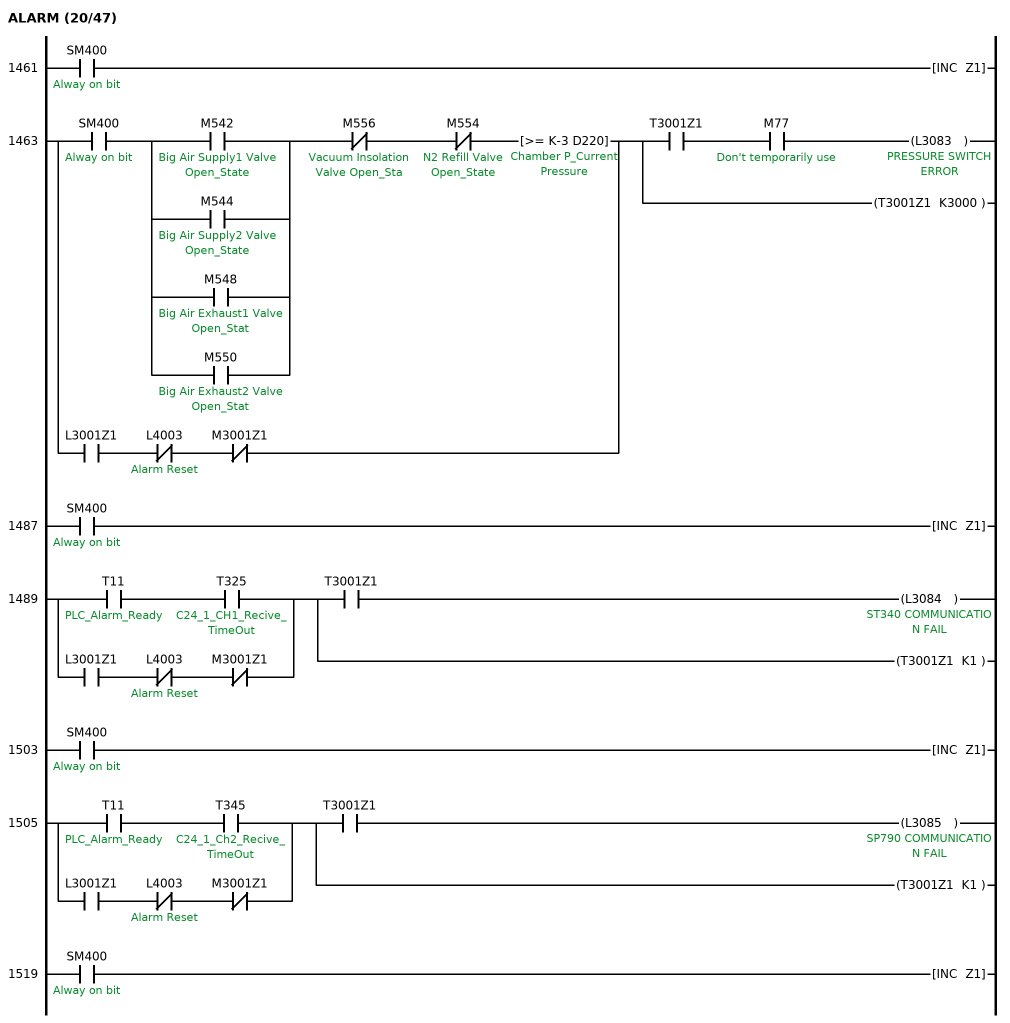
1461  LD      SM400  ; Alway on bit
      INC     Z1
1463  LD      SM400  ; Alway on bit
      LD      M542  ; Big Air Supply1 Valve Open_State
      OR      M544  ; Big Air Supply2 Valve Open_State
      OR      M548  ; Big Air Exhaust1 Valve Open_Stat
      OR      M550  ; Big Air Exhaust2 Valve Open_Stat
      ANB
      ANI     M556  ; Vacuum Insolation Valve Open_Sta
      ANI     M554  ; N2 Refill Valve Open_State
      AND>=   K-3 D220  ; Chamber P_Current Pressure
      LD      L3001Z1
      ANI     L4003  ; Alarm Reset
      ANI     M3001Z1
      ORB
      MPS
      AND     T3001Z1
      AND     M77  ; Don't temporarily use
      OUT     L3083  ; PRESSURE SWITCH ERROR
      MPP
      OUT     T3001Z1 K3000
1487  LD      SM400  ; Alway on bit
      INC     Z1
1489  LD      T11  ; PLC_Alarm_Ready
      AND     T325  ; C24_1_CH1_Recive_TimeOut
      LD      L3001Z1
      ANI     L4003  ; Alarm Reset
      ANI     M3001Z1
      ORB
      MPS
      AND     T3001Z1
      OUT     L3084  ; ST340 COMMUNICATION FAIL
      MPP
      OUT     T3001Z1 K1
1503  LD      SM400  ; Alway on bit
      INC     Z1
1505  LD      T11  ; PLC_Alarm_Ready
      AND     T345  ; C24_1_Ch2_Recive_TimeOut
      LD      L3001Z1
      ANI     L4003  ; Alarm Reset
      ANI     M3001Z1
      ORB
      MPS
      AND     T3001Z1
      OUT     L3085  ; SP790 COMMUNICATION FAIL
      MPP
      OUT     T3001Z1 K1
1519  LD      SM400  ; Alway on bit
      INC     Z1
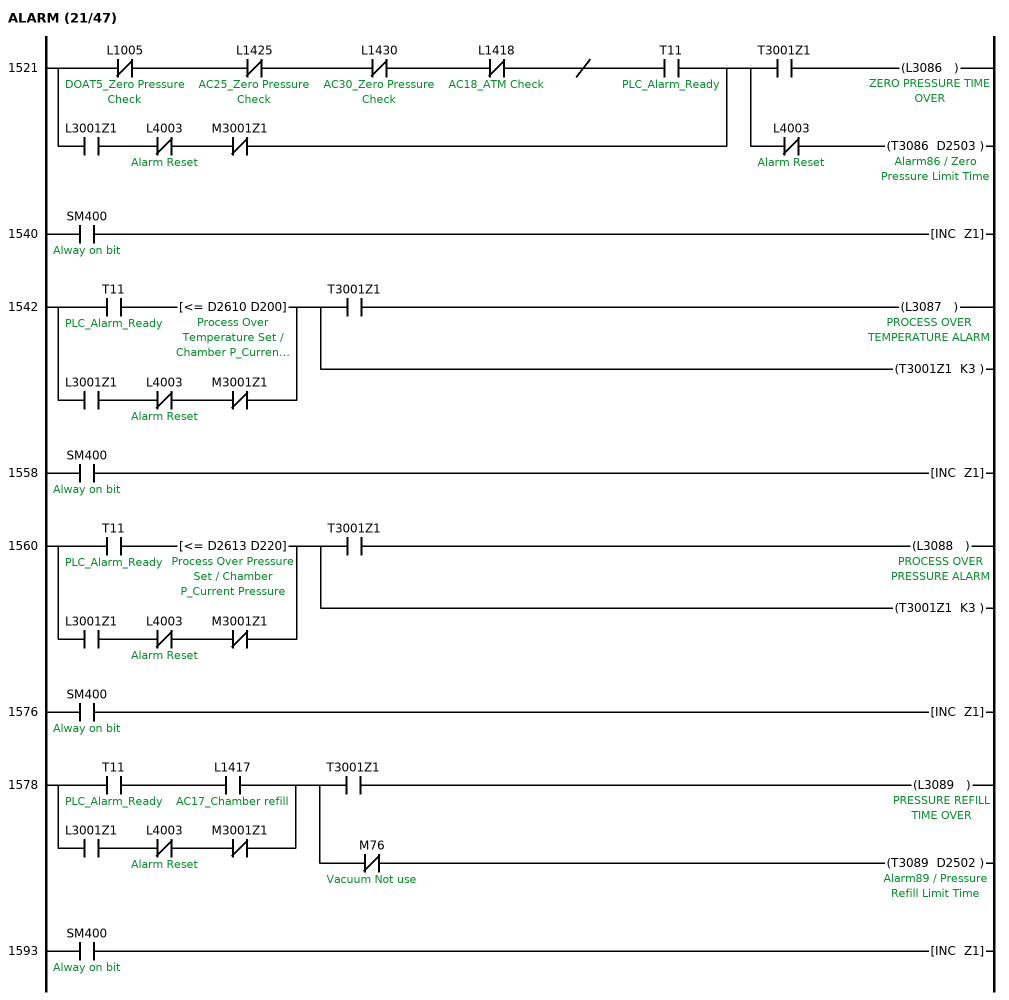
1521  LDI     L1005  ; DOAT5_Zero Pressure Check
      ANI     L1425  ; AC25_Zero Pressure Check
      ANI     L1430  ; AC30_Zero Pressure Check
      ANI     L1418  ; AC18_ATM Check
      INV
      AND     T11  ; PLC_Alarm_Ready
      LD      L3001Z1
      ANI     L4003  ; Alarm Reset
      ANI     M3001Z1
      ORB
      MPS
      AND     T3001Z1
      OUT     L3086  ; ZERO PRESSURE TIME OVER
      MPP
      ANI     L4003  ; Alarm Reset
      OUT     T3086 D2503  ; Alarm86 / Zero Pressure Limit Time
1540  LD      SM400  ; Alway on bit
      INC     Z1
1542  LD      T11  ; PLC_Alarm_Ready
      AND<=   D2610 D200  ; Process Over Temperature Set / Chamber P_Current Temp
      LD      L3001Z1
      ANI     L4003  ; Alarm Reset
      ANI     M3001Z1
      ORB
      MPS
      AND     T3001Z1
      OUT     L3087  ; PROCESS OVER TEMPERATURE ALARM
      MPP
      OUT     T3001Z1 K3
1558  LD      SM400  ; Alway on bit
      INC     Z1
1560  LD      T11  ; PLC_Alarm_Ready
      AND<=   D2613 D220  ; Process Over Pressure Set / Chamber P_Current Pressure
      LD      L3001Z1
      ANI     L4003  ; Alarm Reset
      ANI     M3001Z1
      ORB
      MPS
      AND     T3001Z1
      OUT     L3088  ; PROCESS OVER PRESSURE ALARM
      MPP
      OUT     T3001Z1 K3
1576  LD      SM400  ; Alway on bit
      INC     Z1
1578  LD      T11  ; PLC_Alarm_Ready
      AND     L1417  ; AC17_Chamber refill
      LD      L3001Z1
      ANI     L4003  ; Alarm Reset
      ANI     M3001Z1
      ORB
      MPS
      AND     T3001Z1
      OUT     L3089  ; PRESSURE REFILL TIME OVER
      MPP
      ANI     M76  ; Vacuum Not use
      OUT     T3089 D2502  ; Alarm89 / Pressure Refill Limit Time
1593  LD      SM400  ; Alway on bit
      INC     Z1
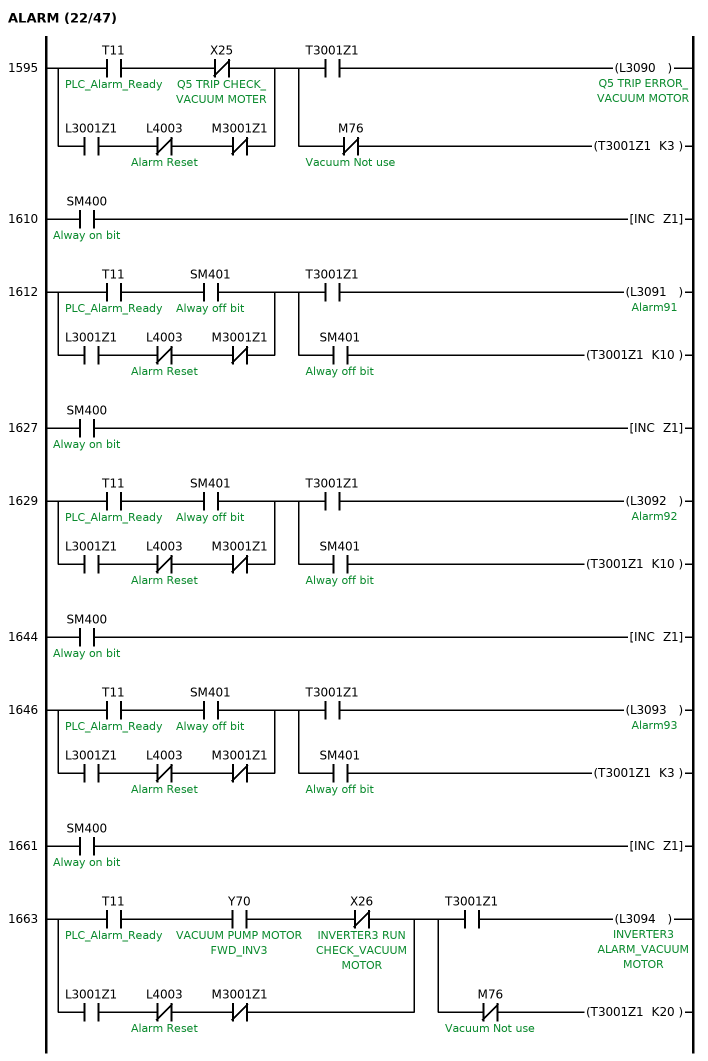
1595  LD      T11  ; PLC_Alarm_Ready
      ANI     X25  ; Q5 TRIP CHECK_VACUUM MOTER
      LD      L3001Z1
      ANI     L4003  ; Alarm Reset
      ANI     M3001Z1
      ORB
      MPS
      AND     T3001Z1
      OUT     L3090  ; Q5 TRIP ERROR_VACUUM MOTOR
      MPP
      ANI     M76  ; Vacuum Not use
      OUT     T3001Z1 K3
1610  LD      SM400  ; Alway on bit
      INC     Z1
1612  LD      T11  ; PLC_Alarm_Ready
      AND     SM401  ; Alway off bit
      LD      L3001Z1
      ANI     L4003  ; Alarm Reset
      ANI     M3001Z1
      ORB
      MPS
      AND     T3001Z1
      OUT     L3091  ; Alarm91
      MPP
      AND     SM401  ; Alway off bit
      OUT     T3001Z1 K10
1627  LD      SM400  ; Alway on bit
      INC     Z1
1629  LD      T11  ; PLC_Alarm_Ready
      AND     SM401  ; Alway off bit
      LD      L3001Z1
      ANI     L4003  ; Alarm Reset
      ANI     M3001Z1
      ORB
      MPS
      AND     T3001Z1
      OUT     L3092  ; Alarm92
      MPP
      AND     SM401  ; Alway off bit
      OUT     T3001Z1 K10
1644  LD      SM400  ; Alway on bit
      INC     Z1
1646  LD      T11  ; PLC_Alarm_Ready
      AND     SM401  ; Alway off bit
      LD      L3001Z1
      ANI     L4003  ; Alarm Reset
      ANI     M3001Z1
      ORB
      MPS
      AND     T3001Z1
      OUT     L3093  ; Alarm93
      MPP
      AND     SM401  ; Alway off bit
      OUT     T3001Z1 K3
1661  LD      SM400  ; Alway on bit
      INC     Z1
1663  LD      T11  ; PLC_Alarm_Ready
      AND     Y70  ; VACUUM PUMP MOTOR FWD_INV3
      ANI     X26  ; INVERTER3 RUN CHECK_VACUUM MOTOR
      LD      L3001Z1
      ANI     L4003  ; Alarm Reset
      ANI     M3001Z1
      ORB
      MPS
      AND     T3001Z1
      OUT     L3094  ; INVERTER3 ALARM_VACUUM MOTOR
      MPP
      ANI     M76  ; Vacuum Not use
      OUT     T3001Z1 K20
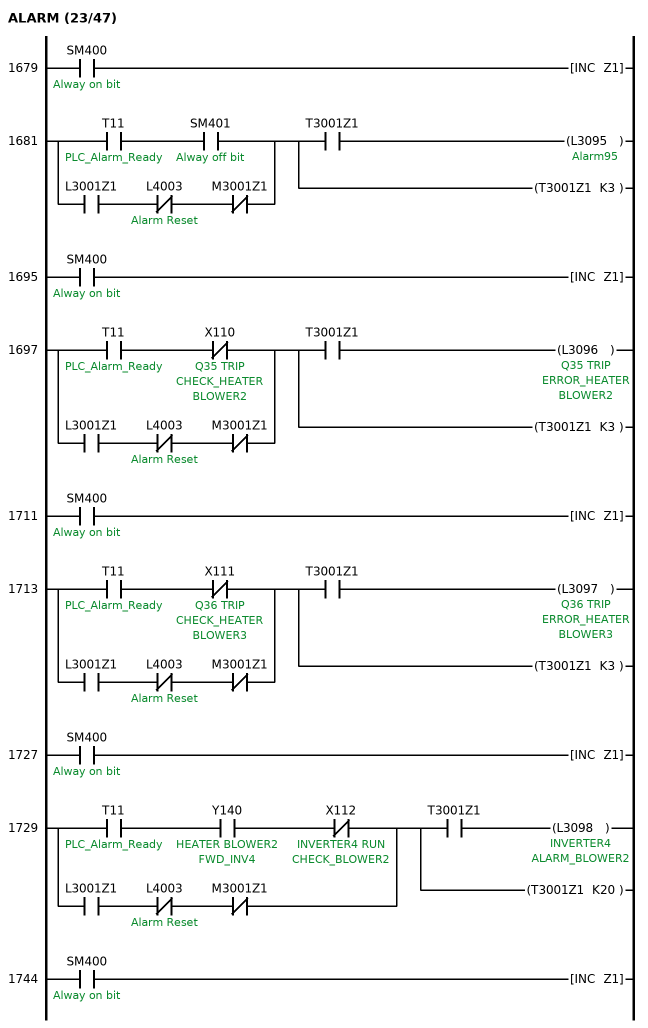
1679  LD      SM400  ; Alway on bit
      INC     Z1
1681  LD      T11  ; PLC_Alarm_Ready
      AND     SM401  ; Alway off bit
      LD      L3001Z1
      ANI     L4003  ; Alarm Reset
      ANI     M3001Z1
      ORB
      MPS
      AND     T3001Z1
      OUT     L3095  ; Alarm95
      MPP
      OUT     T3001Z1 K3
1695  LD      SM400  ; Alway on bit
      INC     Z1
1697  LD      T11  ; PLC_Alarm_Ready
      ANI     X110  ; Q35 TRIP CHECK_HEATER BLOWER2
      LD      L3001Z1
      ANI     L4003  ; Alarm Reset
      ANI     M3001Z1
      ORB
      MPS
      AND     T3001Z1
      OUT     L3096  ; Q35 TRIP ERROR_HEATER BLOWER2
      MPP
      OUT     T3001Z1 K3
1711  LD      SM400  ; Alway on bit
      INC     Z1
1713  LD      T11  ; PLC_Alarm_Ready
      ANI     X111  ; Q36 TRIP CHECK_HEATER BLOWER3
      LD      L3001Z1
      ANI     L4003  ; Alarm Reset
      ANI     M3001Z1
      ORB
      MPS
      AND     T3001Z1
      OUT     L3097  ; Q36 TRIP ERROR_HEATER BLOWER3
      MPP
      OUT     T3001Z1 K3
1727  LD      SM400  ; Alway on bit
      INC     Z1
1729  LD      T11  ; PLC_Alarm_Ready
      AND     Y140  ; HEATER BLOWER2 FWD_INV4
      ANI     X112  ; INVERTER4 RUN CHECK_BLOWER2
      LD      L3001Z1
      ANI     L4003  ; Alarm Reset
      ANI     M3001Z1
      ORB
      MPS
      AND     T3001Z1
      OUT     L3098  ; INVERTER4 ALARM_BLOWER2
      MPP
      OUT     T3001Z1 K20
1744  LD      SM400  ; Alway on bit
      INC     Z1
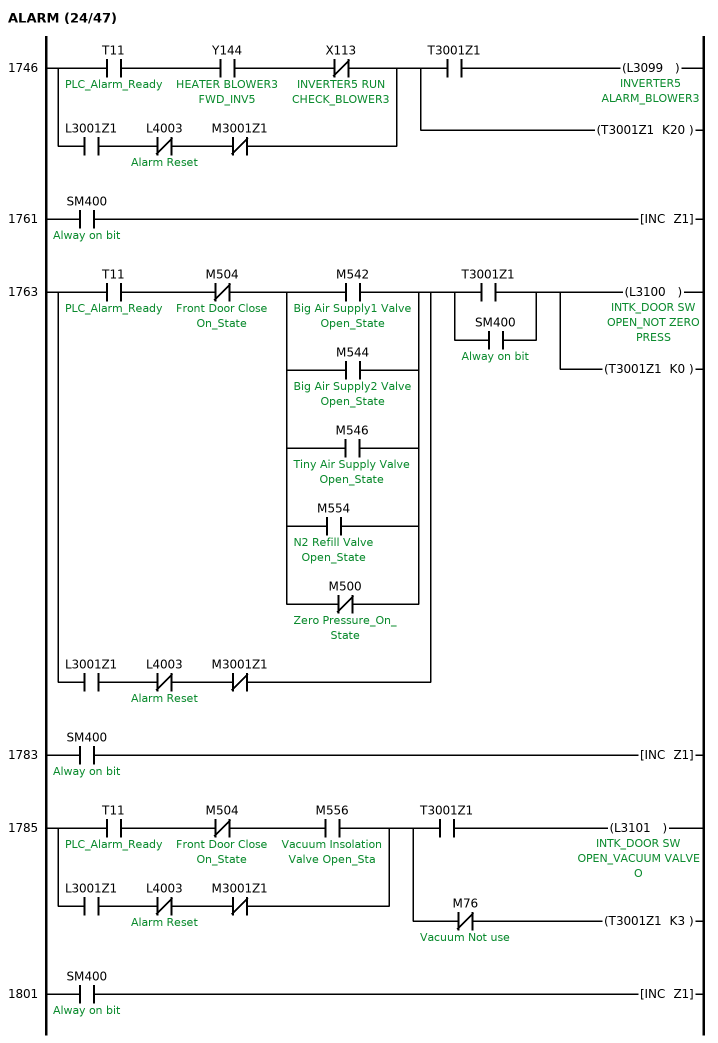
1746  LD      T11  ; PLC_Alarm_Ready
      AND     Y144  ; HEATER BLOWER3 FWD_INV5
      ANI     X113  ; INVERTER5 RUN CHECK_BLOWER3
      LD      L3001Z1
      ANI     L4003  ; Alarm Reset
      ANI     M3001Z1
      ORB
      MPS
      AND     T3001Z1
      OUT     L3099  ; INVERTER5 ALARM_BLOWER3
      MPP
      OUT     T3001Z1 K20
1761  LD      SM400  ; Alway on bit
      INC     Z1
1763  LD      T11  ; PLC_Alarm_Ready
      ANI     M504  ; Front Door Close On_State
      LD      M542  ; Big Air Supply1 Valve Open_State
      OR      M544  ; Big Air Supply2 Valve Open_State
      OR      M546  ; Tiny Air Supply Valve Open_State
      OR      M554  ; N2 Refill Valve Open_State
      ORI     M500  ; Zero Pressure_On_State
      ANB
      LD      L3001Z1
      ANI     L4003  ; Alarm Reset
      ANI     M3001Z1
      ORB
      LD      T3001Z1
      OR      SM400  ; Alway on bit
      ANB
      OUT     L3100  ; INTK_DOOR SW OPEN_NOT ZERO PRESS
      OUT     T3001Z1 K0
1783  LD      SM400  ; Alway on bit
      INC     Z1
1785  LD      T11  ; PLC_Alarm_Ready
      ANI     M504  ; Front Door Close On_State
      AND     M556  ; Vacuum Insolation Valve Open_Sta
      LD      L3001Z1
      ANI     L4003  ; Alarm Reset
      ANI     M3001Z1
      ORB
      MPS
      AND     T3001Z1
      OUT     L3101  ; INTK_DOOR SW OPEN_VACUUM VALVE O
      MPP
      ANI     M76  ; Vacuum Not use
      OUT     T3001Z1 K3
1801  LD      SM400  ; Alway on bit
      INC     Z1
